// TIA Portal V17 export
// export: Created 2022-06-16T09:21:08.1299489Z, ExportSetting WithDefaults, DisplayName Totally Integrated Automation Portal, DisplayVersion V17, DisplayName TIA Portal Openness, DisplayVersion V17, DisplayName TIA Portal Version Control Interface, DisplayVersion V17, DisplayName STEP 7 Professional, DisplayVersion V17, DisplayName STEP 7 Safety, DisplayVersion V17, DisplayName WinCC Advanced, DisplayVersion V17
TYPE "typeMotionControlParam"
// stored: IsFailsafeCompliant false
   STRUCT
      angleInputParam { S7_SetPoint := 'True'} : "typeAngleInputParam";
      remoteInputParam { S7_SetPoint := 'True'} : "typeRemoteInputParam";
      angularSpeedGains : Array[1.."AXIS_NUM"] of Real;
      cartSpeedGains : Array[1.."AXIS_NUM"] of Real;
      regulParams { S7_SetPoint := 'True'} : Array[1.."AXIS_NUM"] of "typeRegulParam";
      outputParam { S7_SetPoint := 'True'} : "typePropOutputParam";
      satParam { S7_SetPoint := 'True'} : "typeSatParam";
      minSetpoint { S7_SetPoint := 'True'} : Real;
      minSpeed : Real;
   END_STRUCT;
END_TYPE
